// TIA Portal V17 export
// export: Created 2023-05-31T09:43:47.5745221Z, ExportSetting WithDefaults, DisplayName Totally Integrated Automation Portal, DisplayVersion V17 Update 3, DisplayName TIA Portal Openness, DisplayVersion V17 Update 3, DisplayName TIA Portal Teamcenter Gateway, DisplayVersion V17 Update 3, DisplayName TIA Portal Version Control Interface, DisplayVersion V17, DisplayName STEP 7 Professional, DisplayVersion V17 Update 3, DisplayName STEP 7 Safety, DisplayVersion V17, DisplayName WinCC UA Professional, DisplayVersion V17 Update 3
DATA_BLOCK "Prova_DB"   // DB1
VERSION : 0.1
// stored: AutoNumber true, DBAccessibleFromOPCUA true, DBAccessibleFromWebserver true, InstanceOfName Prova, InstanceOfType FB
"Prova"
   // VAR_INPUT
   //    Start : Bool;
   // END_VAR
   // VAR_OUTPUT
   //    Alarme : Bool;
   // END_VAR
BEGIN
END_DATA_BLOCK
